FUNCTION_BLOCK FB_EstacionRestaurar_SFC
VAR_INPUT
	 // SFC-Flags
    SFCPause: BOOL;
    SFCReset: BOOL;
    
    // Indicadores de sincronizacion
    Ack: BOOL := TRUE;
    Execute: BOOL;
    
    // Entradas
    DescargadorDetras: BOOL := TRUE; 
END_VAR
VAR_OUTPUT
	 // Indicadores de sincronizacion
    Done: BOOL;
    Ready: BOOL;
    
    // Salidas
    DescargadorAtras: BOOL;
END_VAR
VAR
END_VAR

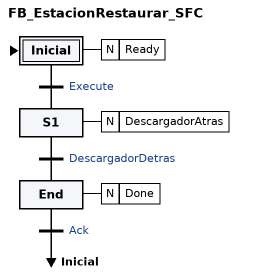
INITIAL_STEP Inicial:
    Ready(N);
END_STEP
TRANSITION FROM Inicial TO S1
    := Execute;
END_TRANSITION
STEP S1:
    DescargadorAtras(N);
END_STEP
TRANSITION FROM S1 TO End
    := DescargadorDetras;
END_TRANSITION
STEP End:
    Done(N);
END_STEP
TRANSITION FROM End TO Inicial
    := Ack;
END_TRANSITION

END_FUNCTION_BLOCK

(* stored: Version 1.1.0.1, ProductVersion 3.1.4024.12
   POU FB_EstacionRestaurar_SFC: Id {7b05be2a-63a0-4839-a320-dfb1a7e175ee}, SpecialFunc None *)
